{attribute 'qualified_only'}
VAR_GLOBAL
	nTemperature AT %I* : INT;
    bInputN1 AT %I* : BOOL;
    bOutputN1 AT %Q* : BOOL;	
END_VAR

(* stored: Version 1.1.0.1
   GVL IO: Id {af4e1bfc-0b35-4beb-bd5d-7e6b1f6827b5} *)
